Yaskawa INFORM job: pneumatic_pod_planes_program.JBI

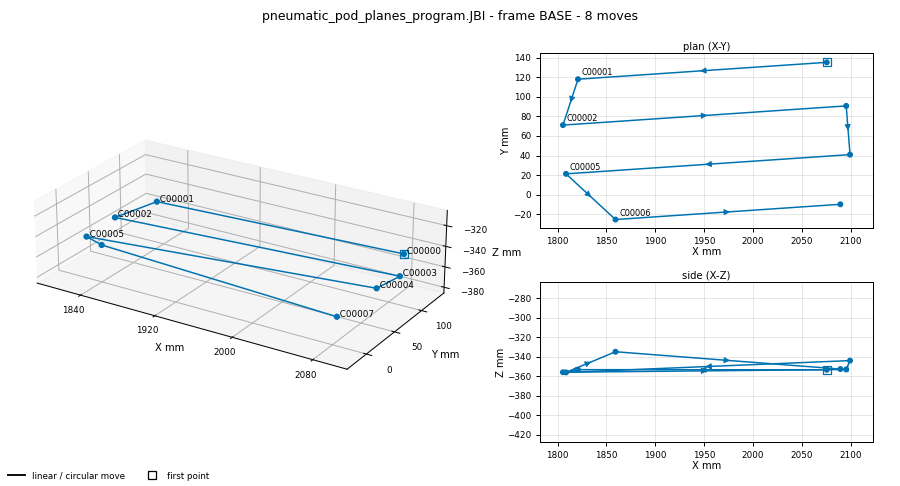
[picture p0: tool path of pneumatic_pod_planes_program.JBI in frame BASE, 8 of 10 moves have a stored position in this frame; points joined in program order, loops and branches not executed]
/JOB
//NAME pneumatic_pod_planes_program
//POS
///NPOS 8,0,8,0,0,0
///TOOL 0
///POSTYPE BASE
///RECTAN
///RCONF 0,0,0,0,0,0,0,0,0,0,0,0,0,0,0,0,0,0,0,0,0,0,0,0
C00000=2075.482830,135.326092,-353.393000,175.000000,-5.000000,5.000000
C00001=1820.900641,118.075262,-353.269967,175.000000,-5.000000,5.000000
C00002=1805.513412,71.112542,-355.912967,175.000000,-5.000000,5.000000
C00003=2095.336099,90.751314,-353.085967,175.000000,-5.000000,5.000000
C00004=2099.262662,40.902725,-343.997967,175.000000,-5.000000,5.000000
C00005=1808.636317,21.209495,-356.063967,175.000000,-5.000000,5.000000
C00006=1859.258686,-25.525038,-334.934967,175.000000,-5.000000,5.000000
C00007=2089.361422,-9.932970,-352.662967,175.000000,-5.000000,5.000000
///POSTYPE PULSE
///PULSE
EC00000=96256.0
EC00001=96256.0
EC00002=96256.0
EC00003=96256.0
EC00004=96256.0
EC00005=96256.0
EC00006=96256.0
EC00007=96256.0
//INST
///DATE 2023/08/16 17:10
///ATTR SC,RW,RJ
////FRAME BASE
///GROUP1 RB1,ST1
NOP
MOVJ P009 EX000 VJ=15.00
MOVJ C00000 EC00000 VJ=15.0
CALL JOB:SPYON
MOVL C00001 EC00001 V=150.0
MOVL C00002 EC00002 V=150.0
MOVL C00003 EC00003 V=150.0
MOVL C00004 EC00004 V=150.0
MOVL C00005 EC00005 V=150.0
MOVL C00006 EC00006 V=150.0
MOVL C00007 EC00007 V=150.0
CALL JOB:SPYOF
MOVJ P009 VJ=15.00
END
